// TIA Portal V20 export
TYPE "LER_typeCommunicationDataS2R"
// stored: Access Published
   STRUCT
      UnitStatus { S7_SetPoint := 'True'} : "LER_typeCommunicationUnitStatus";
      InterfaceData { S7_SetPoint := 'True'} : "LER_typeCommunicationInterfaceData";
   END_STRUCT;
END_TYPE
